Universal Robots PolyScope program: v2ross_teste_comunicacao.urp

Program v2ross_teste_comunicacao (installation=botross directory=/programs/usbdisk/APS2OsUltimosRomanticos createdIn=3.15.3.106223 lastSavedIn=3.15.3.106223 robotSerialNumber=2017357016)
Calibrated DH parameters: a=[0.000147, -0.403633, -0.391058, 0.000042, 0.000118, 0]; d=[0.089178, 30.14366, -33.809995, 3.776935, 0.094786, 0.082481]; alpha=[1.56929, -0.004446, 0.00863, 1.569893, -1.570304, 0]; deltaTheta=[0.000049, -0.320568, 0.239888, 0.08077, 0.000061, 0.000065]
BeforeStart
  'Open Socket that checks if a color is done'
  Socket_color := socket_open("10.103.16.232",30001,socket_name="color")
  'Open Socket that recieve the (X,Y,Z) coordinates data'
  Socket_coord := socket_open("10.103.16.232",30002,socket_name="coord")
  points_done := True
Robot Program (runOnlyOnce=false)
  Loop While (checkContinuously=false) expression=Socket_color ≟  False
    Socket_color := socket_open("10.103.16.232",30001,socket_name="color")
  SuppressedNode
    points_done := socket_read_string(socket_name="color")
  Socket_color := socket_send_string("color_done", socket_name = "color")
  Loop While (checkContinuously=false) expression=Socket_coord ≟ False
    Socket_coord := socket_open("10.103.16.232",30002,socket_name="coord")
  If points_done ≟  False
    Loop While (checkContinuously=false) expression=count≤N
      move2pose := p[X[count]/1000,Y[count]/1000,Z[count]/1000,0,0,0]
      MoveL speed 200 mm/s, acceleration 600 mm/s^2 (useActiveTCP=true) feature=Plano_Pintura
        Waypoint Waypoint (Variable): variable=move2pose
      SuppressedNode
        Wait Sleep waitTime=0.5
      count := count+1
Thread Thread_1 (runOnlyOnce=false)
  points_done := socket_read_string(socket_name="color")
  If points_done ≟ False
    Loop While (checkContinuously=false) expression=(Socket_coord ≟ False )≟ False
      Num_points := socket_read_ascii_float(1,socket_name="coord")
      N := Num_points[1]
      X := socket_read_ascii_float(N,socket_name="coord")
      Y := socket_read_ascii_float(N,socket_name="coord")
      Z := socket_read_ascii_float(N,socket_name="coord")
      count := 1
      ready_to_move := True
  Else 
    ready_to_move := False
    points_done := True
